Fanuc TP program (LS listing): UP021.LS

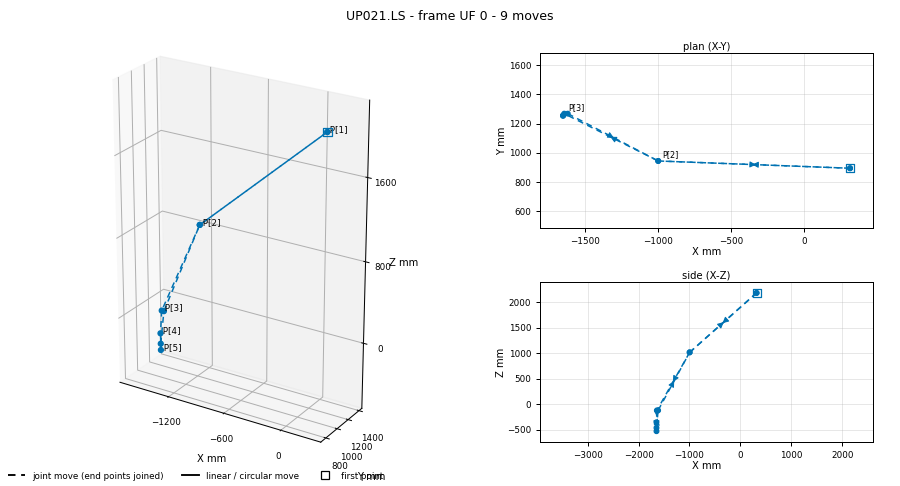
[picture p0: tool path of UP021.LS in frame UF 0, 9 of 9 moves have a stored position in this frame; points joined in program order, loops and branches not executed]
/PROG  UP021
/ATTR
OWNER		= GME;
COMMENT		= "Tomar en ST1620";
PROG_SIZE	= 4398;
CREATE		= DATE 96-03-29  TIME 13:15:26;
MODIFIED	= DATE 24-03-23  TIME 12:09:14;
FILE_NAME	= UP021;
VERSION		= 0;
LINE_COUNT	= 20;
MEMORY_SIZE	= 7926;
PROTECT		= READ_WRITE;
TCD:  STACK_SIZE	= 500,
      TASK_PRIORITY	= 50,
      TIME_SLICE	= 0,
      BUSY_LAMP_OFF	= 0,
      ABORT_REQUEST	= 0,
      PAUSE_REQUEST	= 0;
DEFAULT_GROUP	= 1,1,1,1,*;
CONTROL_CODE	= 00000000 00000000;
/APPL
/MN
   1:  UFRAME_NUM=0 ;
   2:  UTOOL_NUM=1 ;
   3:  PAYLOAD[1] ;
   4:  !Apagar Perfil Lib. 80 vs ST1620 ;
   5:  !Encender Anticol. 1 vs 1610R01 ;
   6:J P[1] 100% CNT0 ACC100 TB    0.00sec,P-SPS    ;
      1:  TC_ONLINE (ON) ;
      2:  DO[23]=OFF ;
      3:  TIMER[3]=RESET ;
      4:  TIMER[3]=START ;
      5:  CALL MAKRO050    ;
      6:  !Lib. de Herramientas ;
      7:  DO[80]=ON ;
      8:  DO[78]=OFF ;
      9:  DO[77]=ON ;
     10:  DO[75]=OFF ;
     11:  !Lib. de Anticolisiones ;
     12:  DO[41]=ON ;
     13:  DO[42]=ON ;
     14:  DO[43]=ON ;
     15:  DO[44]=ON ;
     16:  !Apagar Pos. Base ;
     17:  DO[15]=OFF ;
     18:  !Robot en Trayectoria ;
     19:  DO[16]=ON ;
     20:  WAIT (DI[64] AND !DI[63] AND DI[80] AND M[2] AND M[31] AND M[33])    ;
     21:  DO[80]=OFF ;
     22:  !Encender Anticolisiones ;
     23:  DO[81]=ON ;
     24:  CALL MAKRO020    ;
     25:  WAIT (DI[23])    ;
     26:  DO[23]=ON ;
     27:  TC_ONLINE (DI[41] AND !DI[63] AND DI[64] AND DI[80] AND M[2] AND M[30] AND M[31] AND M[33] AND M[95] AND M[96]) ;
       ------ ;
   7:J P[2] 100% CNT100 ACC100 TB   0.00sec,P-SPS    ;
      1:  TC_ONLINE (DI[41] AND !DI[63] AND DI[64] AND DI[80] AND M[2] AND M[30] AND M[31] AND M[33] AND M[95] AND M[96]) ;
       ------ ;
   8:J P[3] 100% CNT100 ACC100 TB   0.00sec,P-SPS    ;
      1:  TC_ONLINE (DI[41] AND !DI[63] AND DI[64] AND DI[80] AND M[2] AND M[30] AND M[31] AND M[33] AND M[95] AND M[96]) ;
       ------ ;
   9:J P[4] 100% CNT100 ACC100 TB   0.00sec,P-SPS    ;
      1:  TC_ONLINE (DI[41] AND !DI[63] AND DI[64] AND DI[80] AND M[30] AND M[31] AND M[33] AND M[95] AND M[96]) ;
       ------ ;
  10:  !En Posicion ST1620 ;
  11:  !Tomar Pieza en ST1620 ;
  12:  !Fin de Trabajo 1 ;
  13:L P[5] 1500mm/sec CNT0 ACC100 TB    0.00sec,P-SPS    ;
      1:  TC_ONLINE (ON) ;
      2:  DO[23]=(OFF) ;
      3:  WAIT (M[1])    ;
      4:  DO[78]=ON ;
      5:  CALL MAKRO001    ;
      6:  WAIT (DI[79])    ;
      7:  DO[78]=OFF ;
      8:  F[1]=(ON) ;
      9:  CALL MAKRO343    ;
     10:  WAIT (M[32])    ;
     11:  WAIT (DI[23])    ;
     12:  DO[23]=ON ;
     13:  TC_ONLINE (DI[41] AND DI[79] AND M[1] AND M[30] AND M[32] AND M[33] AND M[95] AND M[96]) ;
       ------ ;
  14:  PAYLOAD[2] ;
  15:L P[6] 2000mm/sec CNT100 ACC100 TB   0.00sec,P-SPS    ;
      1:  TC_ONLINE (DI[41] AND DI[63] AND !DI[64] AND DI[79] AND M[1] AND M[30] AND M[32] AND M[33] AND M[95] AND M[96]) ;
       ------ ;
  16:J P[7] 100% CNT100 ACC100 TB   0.00sec,P-SPS    ;
      1:  TC_ONLINE (DI[41] AND DI[63] AND !DI[64] AND DI[79] AND M[1] AND M[30] AND M[32] AND M[33] AND M[95] AND M[96]) ;
       ------ ;
  17:J P[8] 100% CNT100 ACC100 TB   0.00sec,P-SPS    ;
      1:  TC_ONLINE (DI[41] AND DI[63] AND !DI[64] AND DI[79] AND M[1] AND M[30] AND M[32] AND M[33] AND M[95] AND M[96]) ;
       ------ ;
  18:  !Encender Perfil Lib 80 vs ST1620 ;
  19:  !Apagar Anticol. 1 vs 1610R01 ;
  20:J P[9] 100% CNT0 ACC100 TB    .10sec,P-SPS    ;
      1:  TC_ONLINE (ON) ;
      2:  DO[23]=OFF ;
      3:  TIMER[3]=STOP ;
      4:  DO[41]=ON ;
      5:  DO[80]=ON ;
      6:  WAIT (DI[23])    ;
      7:  DO[23]=ON ;
      8:  TC_ONLINE (M[1] AND M[30] AND M[32] AND M[33] AND M[95] AND M[96]) ;
       ------ ;
/POS
P[1]{
   GP1:
	UF : 0, UT : 1,		CONFIG : 'F U T, 0, 1, 0',
	X =   317.191  mm,	Y =   894.705  mm,	Z =  2184.773  mm,
	W =     0.000 deg,	P =    15.000 deg,	R =    90.000 deg
   GP2:
	UF : 0, UT : 1,
	J1=   100.000  mm
   GP3:
	UF : 0, UT : 1,
	J1=     0.000  mm
   GP4:
	UF : 0, UT : 1,
	J1=     0.000  mm
};
P[2]{
   GP1:
	UF : 0, UT : 1,		CONFIG : 'F U T, 0, 1, 0',
	X =  -996.969  mm,	Y =   944.425  mm,	Z =  1017.771  mm,
	W =     -.107 deg,	P =    55.000 deg,	R =   149.883 deg
   GP2:
	UF : 0, UT : 1,
	J1=   100.000  mm
   GP3:
	UF : 0, UT : 1,
	J1=     0.000  mm
   GP4:
	UF : 0, UT : 1,
	J1=     0.000  mm
};
P[3]{
   GP1:
	UF : 0, UT : 1,		CONFIG : 'F U T, 0, 1, 0',
	X = -1640.500  mm,	Y =  1268.601  mm,	Z =  -122.003  mm,
	W =   180.000 deg,	P =    90.000 deg,	R =     0.000 deg
   GP2:
	UF : 0, UT : 1,
	J1=   100.000  mm
   GP3:
	UF : 0, UT : 1,
	J1=     0.000  mm
   GP4:
	UF : 0, UT : 1,
	J1=     0.000  mm
};
P[4]{
   GP1:
	UF : 0, UT : 1,		CONFIG : 'F U T, 0, 1, 0',
	X = -1649.211  mm,	Y =  1254.680  mm,	Z =  -355.372  mm,
	W =   -95.573 deg,	P =    89.949 deg,	R =    84.463 deg
   GP2:
	UF : 0, UT : 1,
	J1=   100.000  mm
   GP3:
	UF : 0, UT : 1,
	J1=     0.000  mm
   GP4:
	UF : 0, UT : 1,
	J1=     0.000  mm
};
P[5]{
   GP1:
	UF : 0, UT : 1,		CONFIG : 'F U T, 0, 1, 0',
	X = -1648.113  mm,	Y =  1255.674  mm,	Z =  -530.486  mm,
	W =   160.338 deg,	P =    89.984 deg,	R =   -20.175 deg
   GP2:
	UF : 0, UT : 1,
	J1=   100.000  mm
   GP3:
	UF : 0, UT : 1,
	J1=     0.000  mm
   GP4:
	UF : 0, UT : 1,
	J1=     0.000  mm
};
P[6]{
   GP1:
	UF : 0, UT : 1,		CONFIG : 'F U T, 0, 0, 0',
	X = -1648.535  mm,	Y =  1255.343  mm,	Z =  -464.244  mm,
	W =   108.933 deg,	P =    89.972 deg,	R =   -71.097 deg
   GP2:
	UF : 0, UT : 1,
	J1=   100.062  mm
   GP3:
	UF : 0, UT : 1,
	J1=     0.000  mm
   GP4:
	UF : 0, UT : 1,
	J1=     0.000  mm
};
P[7]{
   GP1:
	UF : 0, UT : 1,		CONFIG : 'F U T, 0, 1, 0',
	X = -1616.260  mm,	Y =  1268.602  mm,	Z =  -122.004  mm,
	W =   180.000 deg,	P =    90.000 deg,	R =     0.000 deg
   GP2:
	UF : 0, UT : 1,
	J1=   100.000  mm
   GP3:
	UF : 0, UT : 1,
	J1=     0.000  mm
   GP4:
	UF : 0, UT : 1,
	J1=     0.000  mm
};
P[8]{
   GP1:
	UF : 0, UT : 1,		CONFIG : 'F U T, 0, 1, 0',
	X =  -996.969  mm,	Y =   944.425  mm,	Z =  1017.771  mm,
	W =     -.107 deg,	P =    55.000 deg,	R =   149.883 deg
   GP2:
	UF : 0, UT : 1,
	J1=   100.000  mm
   GP3:
	UF : 0, UT : 1,
	J1=     0.000  mm
   GP4:
	UF : 0, UT : 1,
	J1=     0.000  mm
};
P[9]{
   GP1:
	UF : 0, UT : 1,		CONFIG : 'F U T, 0, 1, 0',
	X =   317.190  mm,	Y =   894.706  mm,	Z =  2184.774  mm,
	W =     0.000 deg,	P =    15.000 deg,	R =    90.000 deg
   GP2:
	UF : 0, UT : 1,
	J1=   100.000  mm
   GP3:
	UF : 0, UT : 1,
	J1=     0.000  mm
   GP4:
	UF : 0, UT : 1,
	J1=     0.000  mm
};
/END
